// TIA Portal V20 export
// export: Created 2025-12-01T14:57:06.3367631Z, ExportSetting None, DisplayName Totally Integrated Automation Portal, DisplayVersion V20 Update 3, DisplayName TIA Portal Openness, DisplayVersion V20 Update 3, DisplayName TIA Portal Version Control Interface, DisplayVersion V20 Update 3, DisplayName STEP 7 Professional, DisplayVersion V20 Update 3, DisplayName STEP 7 Safety, DisplayVersion V20 Update 2, DisplayName WinCC Basic/Comfort/Advanced, DisplayVersion V20 Update 3, DisplayName WinCC Professional, DisplayVersion V20 Update 3, DisplayName WinCC Unified, DisplayVersion V20 Update 3
FUNCTION "FC914_SumaTiempo_DT" : Void   // FC914, STL
{ S7_Optimized_Access := 'FALSE' }
// stored: AutoNumber false
   VAR_IN_OUT
      TiempoActual : Time_Of_Day;
   END_VAR
   VAR_TEMP
      TiempoTMP : Date_And_Time;
   END_VAR
BEGIN

NETWORK
TITLE = Suma Time_of_Date + incremento -> Time_of_Date

      CALL  T_COMBINE
      ( IN1 := D#1990-01-01,
        IN2 := #TiempoActual,
        OUT := #TiempoTMP
      );

      CALL  T_ADD
      ( IN1 := #TiempoTMP,
        IN2 := "DB921_DATOS_FECHA_HORA".Incremento_Tiempo,
        OUT := #TiempoTMP
      );

      CALL  T_CONV
      ( IN  := #TiempoTMP,
        OUT := #TiempoActual
      );

END_FUNCTION
